// TIA Portal V18 export
FUNCTION "Reset Error" : Void   // FC15, LAD
{ S7_Optimized_Access := 'TRUE' }
AUTHOR : HenriP
VERSION : 0.1
// stored: AutoNumber true, IsIECCheckEnabled false, SetENOAutomatically false, UDAEnableTagReadback false
   VAR_INPUT
      FestoAxisFault : Bool;
   END_VAR
   VAR_IN_OUT
      ResetCommand : Bool;
      FestoReset : Bool;
   END_VAR
BEGIN

REGION Network 1: Send Reset Command Flip Flop logic on Command
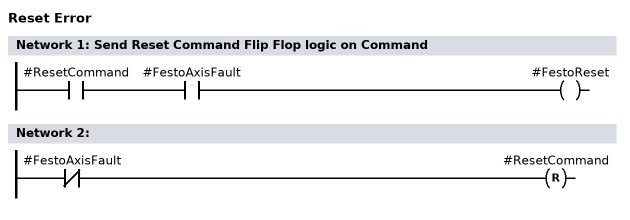
   RUNG wire#powerrail
      Contact( #ResetCommand )
      Contact( #FestoAxisFault )
      Coil( #FestoReset )
   END_RUNG
   // the same network as SCL:
   #FestoReset := #ResetCommand AND #FestoAxisFault;
END_REGION

REGION Network 2
   RUNG wire#powerrail
      I_Contact( #FestoAxisFault )
      R_Coil( #ResetCommand )
   END_RUNG
   // the same network as SCL:
   IF NOT #FestoAxisFault THEN #ResetCommand := FALSE; END_IF;
END_REGION
END_FUNCTION
